SUBAPPLICATION AR_SERVER_0_1_TO_Publish_OPC (* Empfaengt einen REAL-Wert als Argument eines entfernten OPC-UA-Methodenaufrufs (CALL_METHOD, AR_SERVER_0_1) und publiziert ihn sofort lokal weiter (AR_PUBLISH_1) - kein VT-Anschluss, reine Weiterleitungsbruecke fuer Stationen ohne VT. Fuer 'VT-Eingabefeld auf einer anderen Station ODER Web-Dashboard rufen dieselbe Methode auf, nur bei echter Eingabe' (Franz), z.B. Druck-Referenzwerte (B20). *)
  (* Standard: 61499-2; Description: Copyright (c) 2026 Meisterschulen am Ostbahnhof This program and the accompanying materials are made available under the terms of the Eclipse Public License 2.0 which is available at https://www.eclipse.org/legal/epl-2.0/ SPDX-License-Identifier: EPL-2.0 *)
  (* Version 1.0, 2026-09-23, Franz Höpfinger, Meisterschulen am Ostbahnhof, initial implementation - Franz: 'man macht auf STG4 2 METHODEN, die werden aufgerufen: vom Web-Dashboard oder von VT1, und zwar nur wenn jemand was eingibt'. Buendelt AR_SERVER_0_1 (Empfang) + AR_PUBLISH_1 (lokale Weiterleitung), fuer Sensor-Stationen ohne eigene VT (z.B. STG4), die trotzdem echte, editierbare Referenzwerte von einer anderen Station (VT) oder dem Dashboard entgegennehmen sollen. *)
  PACKAGE MyLib::sys;
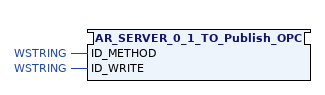
  VAR_INPUT
    ID_METHOD : WSTRING; (* Lokal erzeugte OPC-UA-Methode (ACTION=CREATE_METHOD, 1 REAL-Argument) - von einer anderen Station (AR_CLIENT_1_0) UND/ODER direkt vom OPC-Dashboard aufrufbar *)
    ID_WRITE : WSTRING; (* Lokale Publish-Adresse (REAL, ACTION=PUBLISH) fuer den empfangenen Wert - typischerweise von einem lokalen Self-Subscribe gegengelesen *)
  END_VAR
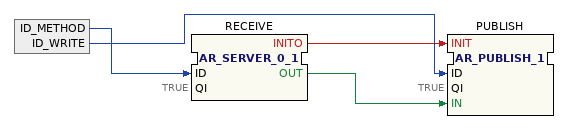
  FBS
    RECEIVE : adapter::net::AR_SERVER_0_1(QI := TRUE);
    PUBLISH : adapter::net::AR_PUBLISH_1(QI := TRUE);
  END_FBS
  EVENT_CONNECTIONS
    RECEIVE.INITO TO PUBLISH.INIT;
  END_CONNECTIONS
  DATA_CONNECTIONS
    ID_METHOD TO RECEIVE.ID;
    ID_WRITE TO PUBLISH.ID;
  END_CONNECTIONS
  ADAPTER_CONNECTIONS
    RECEIVE.OUT TO PUBLISH.IN;
  END_CONNECTIONS
END_SUBAPPLICATION
